INTERFACE ITF_Group2_HMI_Connector EXTENDS
	ITF_BaseGroupElement_HMI_Connector, ITF_Group2_HMI_Connector_View, ITF_Group2_HMI_Connector_Command

END_INTERFACE

(* stored: Version 1.1.0.1
   Itf ITF_Group2_HMI_Connector: Id {8227d0a7-675d-0b56-306c-0f2e82b0b2e6} *)
